// TIA Portal V20 export
VAR_GLOBAL   // PLC tag table "LGR_Const_Equip_TaskStatus"
END_VAR
VAR_GLOBAL CONSTANT   // user constants
   TASK_AWAIT : Byte := 2#0000_0001;   // .X0
   TASK_INPROGRESS : Byte := 2#0000_0010;   // .X1
   TASK_COMPLETE : Byte := 2#0100_0000;   // .X6
   TASK_CANCLED : Byte := 2#1000_0000;   // .X7
END_VAR
